// TwinCAT 3 PLC project SchmittTriggerTests
// ProgramVersion: 3.1.4026.22
// libraries:
//   Tc2_Standard, * (Beckhoff Automation GmbH)
//   Tc2_System, * (Beckhoff Automation GmbH)
//   TcUnit, * (www.tcunit.org)
//   T1SchmittTrigger_Plc,newest,Tc3 Project
// project tree:
//   / PlcTask.TcTTO
//   POUs/ FB_SchmittTriggerConsumer.TcPOU, FB_SchmittTriggerTests.TcPOU, MAIN.TcPOU
// real-time tasks:
//   TASK PlcTask: cycle T#10ms, priority 20, ADS port 350

CONFIGURATION SchmittTriggerTests
    RESOURCE PLC ON TwinCAT3
        TASK PlcTask(INTERVAL := T#10ms, PRIORITY := 20);
        PROGRAM MAIN WITH PlcTask : MAIN;
    END_RESOURCE
END_CONFIGURATION

// ---- POUs/MAIN.TcPOU
PROGRAM MAIN
VAR
    suite : FB_SchmittTriggerTests;
END_VAR

suite();
TcUnit.RUN();

END_PROGRAM

// ---- POUs/FB_SchmittTriggerTests.TcPOU
FUNCTION_BLOCK FB_SchmittTriggerTests EXTENDS TcUnit.FB_TestSuite
VAR
END_VAR

LatchesHighAboveHighThreshold();
LatchesLowBelowLowThreshold();
HoldsInHysteresisBand();
SequencedTransitions();
BoundaryValues();

METHOD PRIVATE BoundaryValues
VAR
    trigger : T1SchmittTrigger_Plc.FB_SchmittTrigger;
    latchedHigh : BOOL;
    atHighBoundary : BOOL;
    afterReset : BOOL;
    atLowBoundary : BOOL;
END_VAR
TEST('BoundaryValues');
trigger(fInput := 0.9);
latchedHigh := trigger.Step();
trigger(fInput := 0.7);
atHighBoundary := trigger.Step();
trigger(fInput := 0.1);
afterReset := trigger.Step();
trigger(fInput := 0.3);
atLowBoundary := trigger.Step();
AssertEquals_BOOL(
    Expected := TRUE,
    Actual := latchedHigh,
    Message := 'fInput := 0.9 should latch HIGH (precondition)');
AssertEquals_BOOL(
    Expected := TRUE,
    Actual := atHighBoundary,
    Message := 'fInput := 0.7 (high boundary, strict >) should hold previous TRUE');
AssertEquals_BOOL(
    Expected := FALSE,
    Actual := afterReset,
    Message := 'fInput := 0.1 should latch LOW (reset for next assertion)');
AssertEquals_BOOL(
    Expected := FALSE,
    Actual := atLowBoundary,
    Message := 'fInput := 0.3 (low boundary, strict <) should hold previous FALSE');
TEST_FINISHED();
END_METHOD

METHOD PRIVATE HoldsInHysteresisBand
VAR
    trigger : T1SchmittTrigger_Plc.FB_SchmittTrigger;
    bResult : BOOL;
END_VAR
TEST('HoldsInHysteresisBand');
trigger(fInput := 0.9);
trigger.Step();
trigger(fInput := 0.5);
bResult := trigger.Step();
AssertEquals_BOOL(
    Expected := TRUE,
    Actual := bResult,
    Message := 'trigger.Step() in band with previous TRUE should hold TRUE');
TEST_FINISHED();
END_METHOD

METHOD PRIVATE LatchesHighAboveHighThreshold
VAR
    trigger : T1SchmittTrigger_Plc.FB_SchmittTrigger;
    bResult : BOOL;
END_VAR
TEST('LatchesHighAboveHighThreshold');
trigger(fInput := 0.9);
bResult := trigger.Step();
AssertEquals_BOOL(
    Expected := TRUE,
    Actual := bResult,
    Message := 'trigger.Step() with fInput := 0.9 should latch HIGH');
TEST_FINISHED();
END_METHOD

METHOD PRIVATE LatchesLowBelowLowThreshold
VAR
    trigger : T1SchmittTrigger_Plc.FB_SchmittTrigger;
    stateHigh : BOOL;
    stateLow : BOOL;
END_VAR
TEST('LatchesLowBelowLowThreshold');
trigger(fInput := 0.9);
stateHigh := trigger.Step();
trigger(fInput := 0.1);
stateLow := trigger.Step();
AssertEquals_BOOL(
    Expected := TRUE,
    Actual := stateHigh,
    Message := 'fInput := 0.9 should first latch HIGH (precondition for LOW test)');
AssertEquals_BOOL(
    Expected := FALSE,
    Actual := stateLow,
    Message := 'fInput := 0.1 (after HIGH) should latch LOW');
TEST_FINISHED();
END_METHOD

METHOD PRIVATE SequencedTransitions
VAR
    trigger : T1SchmittTrigger_Plc.FB_SchmittTrigger;
    state1 : BOOL;
    state2 : BOOL;
    state3 : BOOL;
END_VAR
TEST('SequencedTransitions');
trigger(fInput := 0.5);
state1 := trigger.Step();
trigger(fInput := 0.9);
state2 := trigger.Step();
trigger(fInput := 0.5);
state3 := trigger.Step();
AssertEquals_BOOL(
    Expected := FALSE,
    Actual := state1,
    Message := 'Sequence step 1: 0.5 from default should be FALSE');
AssertEquals_BOOL(
    Expected := TRUE,
    Actual := state2,
    Message := 'Sequence step 2: 0.9 should latch TRUE');
AssertEquals_BOOL(
    Expected := TRUE,
    Actual := state3,
    Message := 'Sequence step 3: 0.5 with previous TRUE should hold TRUE');
TEST_FINISHED();
END_METHOD

END_FUNCTION_BLOCK

// ---- POUs/FB_SchmittTriggerConsumer.TcPOU
FUNCTION_BLOCK FB_SchmittTriggerConsumer
VAR
    trigger : T1SchmittTrigger_Plc.FB_SchmittTrigger;
    bLastState : BOOL;
END_VAR

trigger(fInput := 0.5);
bLastState := trigger.Step();

END_FUNCTION_BLOCK
